{attribute 'linkalways'} 
{attribute 'no_explicit_call' := 'This FB is a CLASS and must be accessed using methods or properties'}
{attribute 'enable_dynamic_creation'}
FUNCTION_BLOCK PUBLIC DefaultGearInBuilder IMPLEMENTS GearInBuilder
VAR
	parent_builder : MotionBuilder;
	parameters : REFERENCE TO DefaultBuilderParameters;
END_VAR

METHOD PUBLIC Acceleration : GearInBuilder
VAR_INPUT
	value : LREAL;
END_VAR
parent_builder.Acceleration(value);
Acceleration := THIS^;
END_METHOD

METHOD PUBLIC BufferMode : GearInBuilder
VAR_INPUT
	mode : MotionBufferMode;
END_VAR
parent_builder.BufferMode(mode);
BufferMode := THIS^;
END_METHOD

METHOD PUBLIC BuildGearInCommand : AsyncCommand
VAR_INPUT
	master_axis : Axis;
	slave_axis : Axis;
END_VAR
VAR
	command_ptr : POINTER TO GearInCommand;
	command : AsyncCommand;
END_VAR
command_ptr := __NEW(GearInCommand(
	master_axis := master_axis,
	slave_axis := slave_axis,
	numerator := parameters.ratio_numerator,
	denominator := parameters.ratio_denominator
// 	deceleration := parameters.deceleration,
// 	jerk := parameters.jerk,
// 	buffer_mode := parameters.buffer_mode
));
BuildGearInCommand := command_ptr^;
END_METHOD

METHOD PUBLIC Deceleration : GearInBuilder
VAR_INPUT
	value : LREAL;
END_VAR
parent_builder.Deceleration(value);
Deceleration := THIS^;
END_METHOD

METHOD Denominator : GearInBuilder
VAR_INPUT
	value : UINT;
END_VAR
parent_builder.Denominator(value);
Denominator := THIS^;
END_METHOD

//FB_Init is always available implicitly and it is used primarily for initialization.
//The return value is not evaluated. For a specific influence, you can also declare the
//methods explicitly and provide additional code there with the standard initialization
//code. You can evaluate the return value.
METHOD FB_Init: BOOL
VAR_INPUT
    bInitRetains : BOOL; // TRUE: the retain variables are initialized (reset warm / reset cold)
    bInCopyCode : BOOL;  // TRUE: the instance will be copied to the copy code afterward (online change)
	parent_builder : MotionBuilder;
	parameters : REFERENCE TO DefaultBuilderParameters;
END_VAR
THIS^.parent_builder := parent_builder;
THIS^.parameters REF= parameters;
END_METHOD

METHOD PUBLIC Jerk : GearInBuilder
VAR_INPUT
	value : LREAL;
END_VAR
parent_builder.Jerk(value);
Jerk := THIS^;
END_METHOD

METHOD Numerator : GearInBuilder
VAR_INPUT
	value : LREAL;
END_VAR
parent_builder.Numerator(value);
Numerator := THIS^;
END_METHOD

METHOD PUBLIC Reset : GearInBuilder
parent_builder.Reset();
Reset := THIS^;
END_METHOD

END_FUNCTION_BLOCK

(* stored: Version 1.1.0.1
   POU DefaultGearInBuilder: Id {212cf965-b7c1-4383-86ef-3a65dc1d2451}, SpecialFunc None
   Folder Builders: Id {72fe9b7c-c2aa-49d3-ac4a-02868f1bc328}
   Folder Constructor: Id {b1076fcb-a73d-4e53-92b1-3fb815d7db3d}
   Folder PropertySetters: Id {0b15a9ed-0629-413d-91e9-daf95a0082be}
   Method Acceleration: Id {7bab9b14-43b5-4d02-b321-0c028237cf78}
   Method BufferMode: Id {ff03d52e-de7f-4997-b3a2-a81177243076}
   Method BuildGearInCommand: Id {26f7a18f-b7a2-4ae9-8cc2-3b63d5f66dca}
   Method Deceleration: Id {11d6416e-405c-4adb-87d3-5c8c03f96f47}
   Method Denominator: Id {a064103a-9f48-4f01-a3db-3bc5357139f9}
   Method FB_Init: Id {df11c2a3-7de9-4dfc-9ec5-21fa31be91f8}
   Method Jerk: Id {b78bf362-1583-47a6-9535-ee8109063b04}
   Method Numerator: Id {a138d0e2-b3ce-4048-be0b-19caa30bfd77}
   Method Reset: Id {7818dd78-3afd-491d-b0dc-f792ab891978} *)
